FUNCTION_BLOCK FB_FieldCodecString IMPLEMENTS I_FieldCodec
VAR_INPUT
END_VAR
VAR_OUTPUT
END_VAR
VAR
    sValue      	: T_MAXSTRING;
    anyStringTmp : T_AnyString;
END_VAR

{attribute 'analysis' := '-33'}
METHOD CalculatePackedDataSize : HRESULT
VAR_INPUT CONSTANT
	anyFirstElem	: T_Any;
	nLength	        : UDINT;        // items to write
END_VAR
VAR_OUTPUT
    nPackedDataSize : UDINT;
END_VAR

CalculatePackedDataSize := 0;
END_METHOD

METHOD IsPackedRepeatedField : BOOL
VAR_INPUT
    {attribute 'analysis' := '-33' } 
	nTag	: UDINT;
END_VAR

IsPackedRepeatedField := FALSE;
END_METHOD

// Needs to be called, if destination string is larger then T_MAXSTRING.
METHOD INTERNAL SetTmpBuffer
VAR_INPUT
    anyString : T_AnyString;
END_VAR
anyStringTmp := anyString;
END_METHOD


METHOD ValueReader : HRESULT
VAR_IN_OUT CONSTANT
	aBuffer	: ARRAY [*] OF BYTE;
END_VAR
VAR_IN_OUT
	stState	: ST_ParserInternalState;
END_VAR
VAR_OUTPUT
	anyOut	: T_Any;
END_VAR
IF anyStringTmp.pValue <> NULL THEN
    anyOut := anyStringTmp;
ELSE
    anyOut := F_ToAnyString(sValue);
END_IF
ValueReader := F_ReadString(aBuffer, stState, anyOut);
END_METHOD

METHOD ValueWriter : HRESULT
VAR_IN_OUT
	aBuffer	: ARRAY [*] OF BYTE;
END_VAR
VAR_IN_OUT
	stState	: ST_WriterInternalState;
END_VAR
VAR_INPUT
    anyIn : T_ANY;
END_VAR

ValueWriter := F_WriteRawString(aBuffer, stState, anyIn);
END_METHOD

END_FUNCTION_BLOCK

(* stored: Version 1.1.0.1
   POU FB_FieldCodecString: Id {15d0b902-f3bf-497f-af92-b61f3894a3cd}, SpecialFunc None
   Method CalculatePackedDataSize: Id {42c73b18-08c1-405a-b45d-edb5b8446815}
   Method IsPackedRepeatedField: Id {eabe9cc3-e78f-42f1-b498-34540e7e1164}
   Method SetTmpBuffer: Id {63850f38-d71f-4abc-b609-7a4032dbd758}
   Method ValueReader: Id {0b25c717-69b6-4051-b2bf-19d82a7ef48c}
   Method ValueWriter: Id {abfdac70-fd08-4671-ada6-743506bccff6} *)
